// TIA Portal V21 export
VAR_GLOBAL   // PLC tag table "Outputs"
   DQ_ColumnRed AT %Q0.0 : Bool;   //    {ExternalWritable false}
   DQ_ColumnGreen AT %Q0.1 : Bool;   //    {ExternalWritable false}
   DQ_Contactor_Pump1 AT %Q0.2 : Bool;   //    {ExternalWritable false}
   DQ_Softstart_Pump1 AT %Q0.3 : Bool;   //    {ExternalWritable false}
   DQ_Contactor_Pump2 AT %Q0.4 : Bool;   //    {ExternalWritable false}
   DQ_Softstart_Pump2 AT %Q0.5 : Bool;   //    {ExternalWritable false}
   DQ_Reserve_0_6 AT %Q0.6 : Bool;   //    {ExternalWritable false}
   DQ_Reserve_0_7 AT %Q0.7 : Bool;   //    {ExternalWritable false}
END_VAR
